// SIMATIC S7-200 project (STEP 7-Micro/WIN), CPU 224XP REL 02.01

SYMBOL_TABLE USUARIO1
PARO             I0.0
MARCHA           I0.1
LAMPARA_1        Q0.0
LAMPARA_2        Q0.1
END_SYMBOL_TABLE

ORGANIZATION_BLOCK PRINCIPAL:OB1
TITLE=COMENTARIOS DEL PROGRAMA
BEGIN
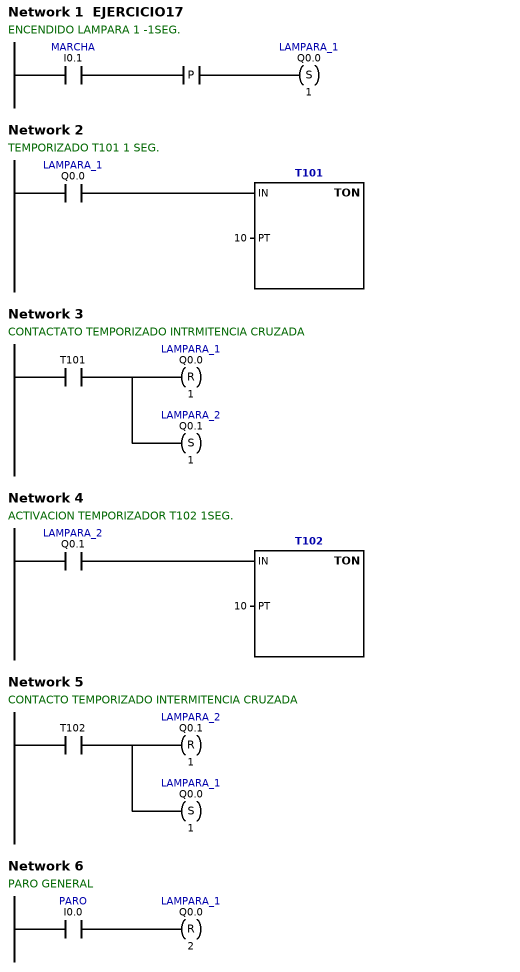
Network 1 // EJERCICIO17
// ENCENDIDO LAMPARA 1 -1SEG.
LD     MARCHA:I0.1
EU
S      LAMPARA_1:Q0.0, 1
Network 2
// TEMPORIZADO T101 1 SEG.
LD     LAMPARA_1:Q0.0
TON    T101, 10
Network 3
// CONTACTATO TEMPORIZADO INTRMITENCIA CRUZADA
LD     T101
R      LAMPARA_1:Q0.0, 1
S      LAMPARA_2:Q0.1, 1
Network 4
// ACTIVACION TEMPORIZADOR T102 1SEG.
LD     LAMPARA_2:Q0.1
TON    T102, 10
Network 5
// CONTACTO TEMPORIZADO INTERMITENCIA CRUZADA
LD     T102
R      LAMPARA_2:Q0.1, 1
S      LAMPARA_1:Q0.0, 1
Network 6
// PARO GENERAL
LD     PARO:I0.0
R      LAMPARA_1:Q0.0, 2
END_ORGANIZATION_BLOCK
